// Mitsubishi GX Works2 project: SetRstY0   PLC: Q03UDV

PROGRAM MAIN
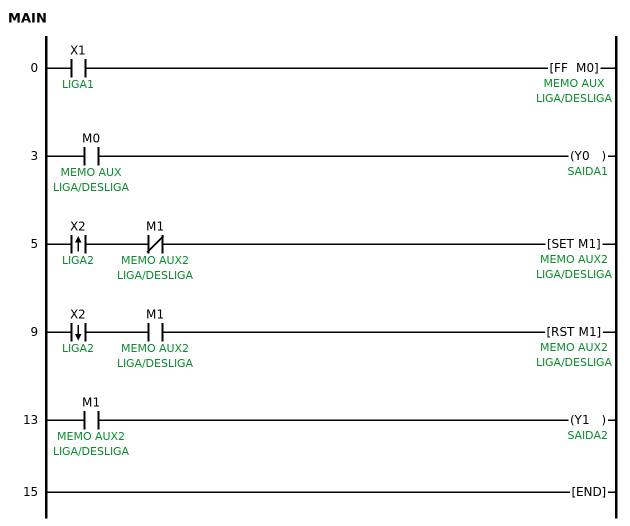
0     LD      X1  ; LIGA1
      FF      M0  ; MEMO AUX LIGA/DESLIGA
3     LD      M0  ; MEMO AUX LIGA/DESLIGA
      OUT     Y0  ; SAIDA1
5     LDP     X2  ; LIGA2
      ANI     M1  ; MEMO AUX2 LIGA/DESLIGA
      SET     M1  ; MEMO AUX2 LIGA/DESLIGA
9     LDF     X2  ; LIGA2
      AND     M1  ; MEMO AUX2 LIGA/DESLIGA
      RST     M1  ; MEMO AUX2 LIGA/DESLIGA
13    LD      M1  ; MEMO AUX2 LIGA/DESLIGA
      OUT     Y1  ; SAIDA2
15    END
END_PROGRAM
